// TwinCAT 3 PLC project PRG_B_ActuatorDecorator
// Title: B_ActuatorDecorator
// Company: RafalOS
// Author: Rafał Osajda
// ProjectVersion: 0.0.0.4
// ProgramVersion: 3.1.4024.0
// libraries:
//   B_Actuator, * (RafalOS)
//   B_Base, * (RafalOS)
//   B_BaseDecorate, * (RafalOS)
//   B_IO, * (RafalOS)
//   B_IODecorator, * (RafalOS)
//   Tc2_Standard, * (Beckhoff Automation GmbH)
//   Tc2_System, * (Beckhoff Automation GmbH)
//   Tc3_Module, * (Beckhoff Automation GmbH)
// project tree:
//   / PlcTask.TcTTO (not stored)
//   POUs Compilation/ PRG_Compilation.TcPOU (not stored)
//   POUs/ FB_Actuator_TestDecorator.TcPOU (not stored), FB_Actuator_TestWithoutTimeDecorator.TcPOU (not stored), FB_Actuator_TestWithTimeDecorator.TcPOU, ITF_ActuatorDecoratorTest.TcIO

// ---- POUs/ITF_ActuatorDecoratorTest.TcIO
INTERFACE ITF_ActuatorDecoratorTest EXTENDS ITF_Actuator

END_INTERFACE

// ---- POUs/FB_Actuator_TestWithTimeDecorator.TcPOU
FUNCTION_BLOCK FB_Actuator_TestWithTimeDecorator EXTENDS FB_Actuator_TestDecorator
VAR
	tonSensorTurnOffTime	: Tc2_Standard.TON;
	tonSensorTurnOnTime		: Tc2_Standard.TON;

END_VAR

(*			
	EVERDE sp. z o.o.
	Rafał Osajda		27.03.2025		TC 4024.66
	Wywolanie co cykl operacji 
*)
METHOD PUBLIC ExecuteEveryCycle_Operation
VAR_INPUT
END_VAR
//testować czy jest cykl przesuwania do gdzieś i po czasie uruchamiać lub wyłączać czujniki 
THIS^.itfactActuator.ExecuteEveryCycle_Operation();
THIS^.tonSensorTurnOffTime ();
THIS^.tonSensorTurnOnTime ();

IF (THIS^.itfactActuator.MovingToStartFirstCycle ()) THEN
	THIS^.itfczStart			:= THIS^.itfsenEnd;
	THIS^.itfczStop				:= THIS^.itfsenStart;
	THIS^.tonSensorTurnOffTime.PT	:= REAL_TO_TIME (THIS^.itfactActuator.ParameterGetValue (1) * 0.1);
	THIS^.tonSensorTurnOffTime.IN	:= TRUE;
	THIS^.tonSensorTurnOnTime.PT	:= REAL_TO_TIME (THIS^.itfactActuator.ParameterGetValue (1) * 0.7);
	THIS^.iStepTestCycle		:= 10;
END_IF

IF (THIS^.itfactActuator.MovingToEndFirstCycyle ()) THEN
	THIS^.itfczStart			:= THIS^.itfsenStart;
	THIS^.itfczStop				:= THIS^.itfsenEnd;
	THIS^.tonSensorTurnOffTime.PT	:= REAL_TO_TIME (THIS^.itfactActuator.ParameterGetValue (2) * 0.1);
	THIS^.tonSensorTurnOffTime.IN	:= TRUE;
	THIS^.tonSensorTurnOnTime.PT	:= REAL_TO_TIME (THIS^.itfactActuator.ParameterGetValue (2) * 0.7);
	THIS^.iStepTestCycle		:= 10;
END_IF

CASE THIS^.iStepTestCycle OF
10	: IF (THIS^.tonSensorTurnOffTime.Q) THEN
		THIS^.tonSensorTurnOffTime.IN	:= FALSE;
		THIS^.itfczStart.SetContact (bIN := FALSE);
		THIS^.tonSensorTurnOnTime.IN	:= TRUE;
		iStepTestCycle		:= THIS^.iStepTestCycle + 10;
	END_IF
20	: IF (THIS^.tonSensorTurnOnTime.Q) THEN
		THIS^.tonSensorTurnOnTime.IN	:= FALSE;
		THIS^.itfczStop.SetContact (bIN := TRUE);
		THIS^.iStepTestCycle	:= 0;
	END_IF
END_CASE
END_METHOD

END_FUNCTION_BLOCK
